% RSLogix 500 project PROJECT_BAK027.RSS, saved by version 8.10.00.18 %
PROJECT "UNTITLED"    % processor: MicroLogix 1400 %

PROGRAM FILES
  LAD 2   19 rungs

DATA FILES
  O0 OUTPUT  6 elements
  I1 INPUT  8 elements
  S2 STATUS  66 elements
  B3 BINARY  2 elements
  T4 TIMER  8 elements
  C5 COUNTER  1 elements
  R6 CONTROL  1 elements
  N7 INTEGER  1 elements
  F8 FLOAT  1 elements

LADDER 2
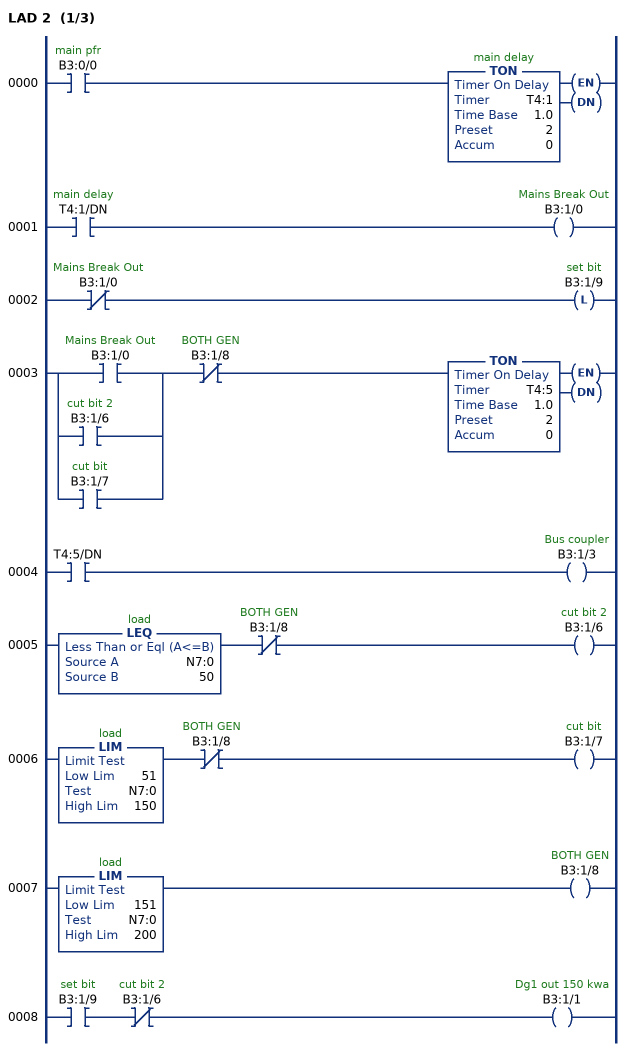
% Rung: 0 %
SOR XIC B3:0/0 TON T4:1 1.0 2 0 EOR
%   B3:0/0  "main pfr" %
%   T4:1  "main delay" %
% Rung: 1 %
SOR XIC T4:1/DN OTE B3:1/0 EOR
%   T4:1  "main delay" %
%   B3:1/0  "Mains Break Out" %
% Rung: 2 %
SOR XIO B3:1/0 OTL B3:1/9 EOR
%   B3:1/0  "Mains Break Out" %
%   B3:1/9  "set bit" %
% Rung: 3 %
SOR BST XIC B3:1/0 NXB BST XIC B3:1/6 NXB XIC B3:1/7 BND BND XIO B3:1/8 TON T4:5 1.0 2 0 EOR
%   B3:1/0  "Mains Break Out" %
%   B3:1/6  "cut bit 2" %
%   B3:1/7  "cut bit" %
%   B3:1/8  "BOTH GEN" %
% Rung: 4 %
SOR XIC T4:5/DN OTE B3:1/3 EOR
%   B3:1/3  "Bus coupler" %
% Rung: 5 %
SOR LEQ N7:0 50 XIO B3:1/8 OTE B3:1/6 EOR
%   N7:0  "load" %
%   B3:1/8  "BOTH GEN" %
%   B3:1/6  "cut bit 2" %
% Rung: 6 %
SOR LIM 51 N7:0 150 XIO B3:1/8 OTE B3:1/7 EOR
%   N7:0  "load" %
%   B3:1/8  "BOTH GEN" %
%   B3:1/7  "cut bit" %
% Rung: 7 %
SOR LIM 151 N7:0 200 OTE B3:1/8 EOR
%   N7:0  "load" %
%   B3:1/8  "BOTH GEN" %
% Rung: 8 %
SOR XIC B3:1/9 XIO B3:1/6 OTE B3:1/1 EOR
%   B3:1/9  "set bit" %
%   B3:1/6  "cut bit 2" %
%   B3:1/1  "Dg1 out 150 kwa" %

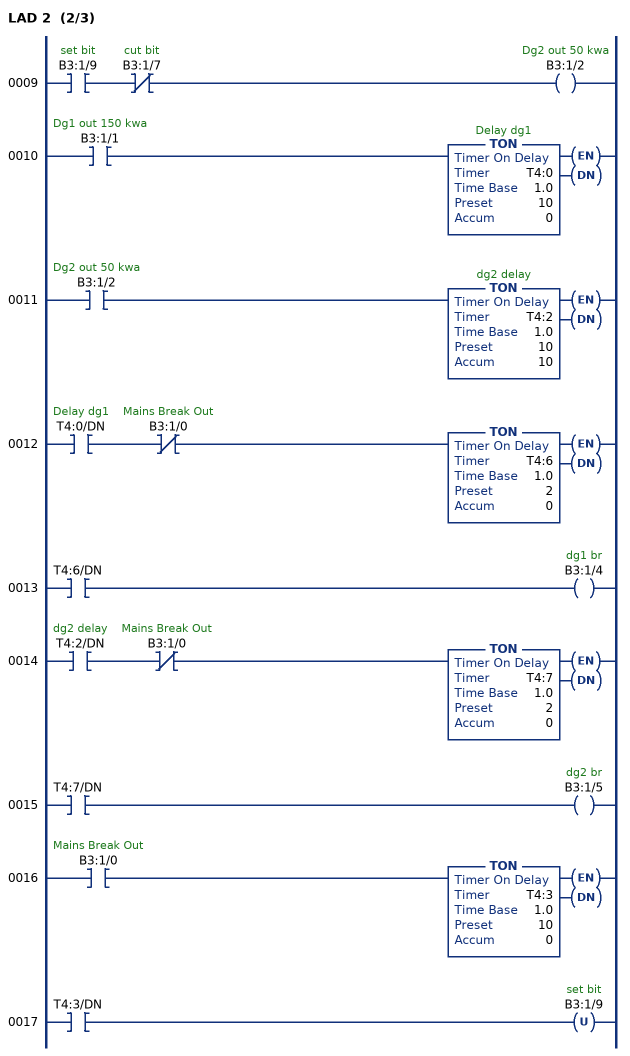
% Rung: 9 %
SOR XIC B3:1/9 XIO B3:1/7 OTE B3:1/2 EOR
%   B3:1/9  "set bit" %
%   B3:1/7  "cut bit" %
%   B3:1/2  "Dg2 out 50 kwa" %
% Rung: 10 %
SOR XIC B3:1/1 TON T4:0 1.0 10 0 EOR
%   B3:1/1  "Dg1 out 150 kwa" %
%   T4:0  "Delay dg1" %
% Rung: 11 %
SOR XIC B3:1/2 TON T4:2 1.0 10 10 EOR
%   B3:1/2  "Dg2 out 50 kwa" %
%   T4:2  "dg2 delay" %
% Rung: 12 %
SOR XIC T4:0/DN XIO B3:1/0 TON T4:6 1.0 2 0 EOR
%   T4:0  "Delay dg1" %
%   B3:1/0  "Mains Break Out" %
% Rung: 13 %
SOR XIC T4:6/DN OTE B3:1/4 EOR
%   B3:1/4  "dg1 br" %
% Rung: 14 %
SOR XIC T4:2/DN XIO B3:1/0 TON T4:7 1.0 2 0 EOR
%   T4:2  "dg2 delay" %
%   B3:1/0  "Mains Break Out" %
% Rung: 15 %
SOR XIC T4:7/DN OTE B3:1/5 EOR
%   B3:1/5  "dg2 br" %
% Rung: 16 %
SOR XIC B3:1/0 TON T4:3 1.0 10 0 EOR
%   B3:1/0  "Mains Break Out" %
% Rung: 17 %
SOR XIC T4:3/DN OTU B3:1/9 EOR
%   B3:1/9  "set bit" %

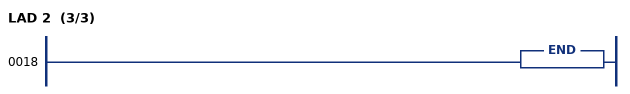
% Rung: 18 %
SOR END EOR

DATA TABLE (non-zero values as saved)
DATA B3
% B3:0 % 0X0000 0X0064
DATA T4
% .PRE .ACC %
% T4:0 % 10 0
% T4:1 % 2 0
% T4:2 % 10 10
% T4:3 % 10 0
% T4:5 % 2 0
% T4:6 % 2 0
% T4:7 % 2 0
DATA N7
% N7:0 % 30
